FUNCTION_BLOCK FB_Blink		// Blink at the specified time
VAR_INPUT
	iTime:		TIME;		// Blinking time
END_VAR
VAR_OUTPUT
	oBlink:		BOOL;		// The blinker (iTime TRUE followed by iTime FALSE)
END_VAR
VAR
	ton:		TON;
	tof: 		TOF;
END_VAR

ton(IN := NOT (oBlink), PT := iTime);
tof(IN := ton.Q, PT := iTime, Q => oBlink);

END_FUNCTION_BLOCK

(* stored: Version 1.1.0.1, ProductVersion 3.1.4026.18
   POU FB_Blink: Id {4e6d1302-a27d-49de-b207-85db729200c0}, SpecialFunc None *)
